PROGRAM GL1_Transfer_Traverse
VAR
	TON_GL1_MTR: TON; // MOTOR FAULT DELAY TIMER
	GL1_MTR: sClearPath;
	GL1_Pulses: INT; // CURRENT PULSE COUNT VALUE
	GL1_Pulse_Counter: CTU; // GL1 MOTOR PULSE COUNTER
	TEST: BOOL;
	GL1_RD: SRoll_Door;
	GL1_PULSE_RESET : BOOL; // RESET THE PULSE COUNTER WHEN COUNTER REACHES PRESET VALUE
	RUN_FWD_TO_GL6_BIT : BOOL; // GL2 OCCUPIED, GL6 REQUESTING PART, RUN TO GL6 POSITION
	RUN_FWD_TO_GL8_BIT : BOOL; // GL2 OCCUPIED, GL8 REQUESTING PART, RUN TO GL8 POSITION
	RUN_REV_TO_GL5B_BIT : BOOL; //GL2 EMPTY, GL2 REQUESTING PART, RUN TO GL5 POSITION
	FAULT_PRESET_TIME: TIME; // FAULT TIMER PRESET TO MOTOR FAULT. DEFAULT IS 1000mS.
	COUNTER_PRESET: WORD; // MAX COUNT VALUE
	TON_GL1_MTR_DONE: BOOL; // TIMER DONE BIT
	KIRK_BIT: BOOL;
	KIRK_BIT2: BOOL;
	KIRK_BIT3: BOOL;
	HI_SPEED: BOOL; // RUN AT HI SPPED TILL FIRST PROX SEEN
	CREEP_SPEED: BOOL; // RUN AT CREEP SPEED TILL SECOND PROX SEEN
	PROX_1_SEEN_AT_GL6: BOOL; // FIRST PROX MADE
	PROX_2_SEEN_AT_GL6: BOOL; // SECOND PROX MADE
	PROX_1_SEEN_AT_GL8: BOOL; // FIRST PROX MADE
	PROX_2_SEEN_AT_GL8: BOOL; // SECOND PROX MADE
	PROX_1_SEEN_AT_GL5B: BOOL; // FIRST PROX MADE
	PROX_2_SEEN_AT_GL5B: BOOL; // SECOND PROX MADE
	TON_CREEP_DELAY: TON; // DELAY CREEP SPEED
	GL6_ENTRY_FTRIG:  F_TRIG;
	GL8_ENTRY_FTRIG:  F_TRIG;
	SwitchFaultTimer: ton;
	SwitchFault: BOOL;
	SwitchTimeElapsed: TIME;
	
END_VAR
VAR // added by the converter: edge detectors and wires of the graphical bodies
    _rt1, _rt2 : R_TRIG;
    _w1, _w2, _w3, _w4, _w5, _w6 : BOOL;
END_VAR

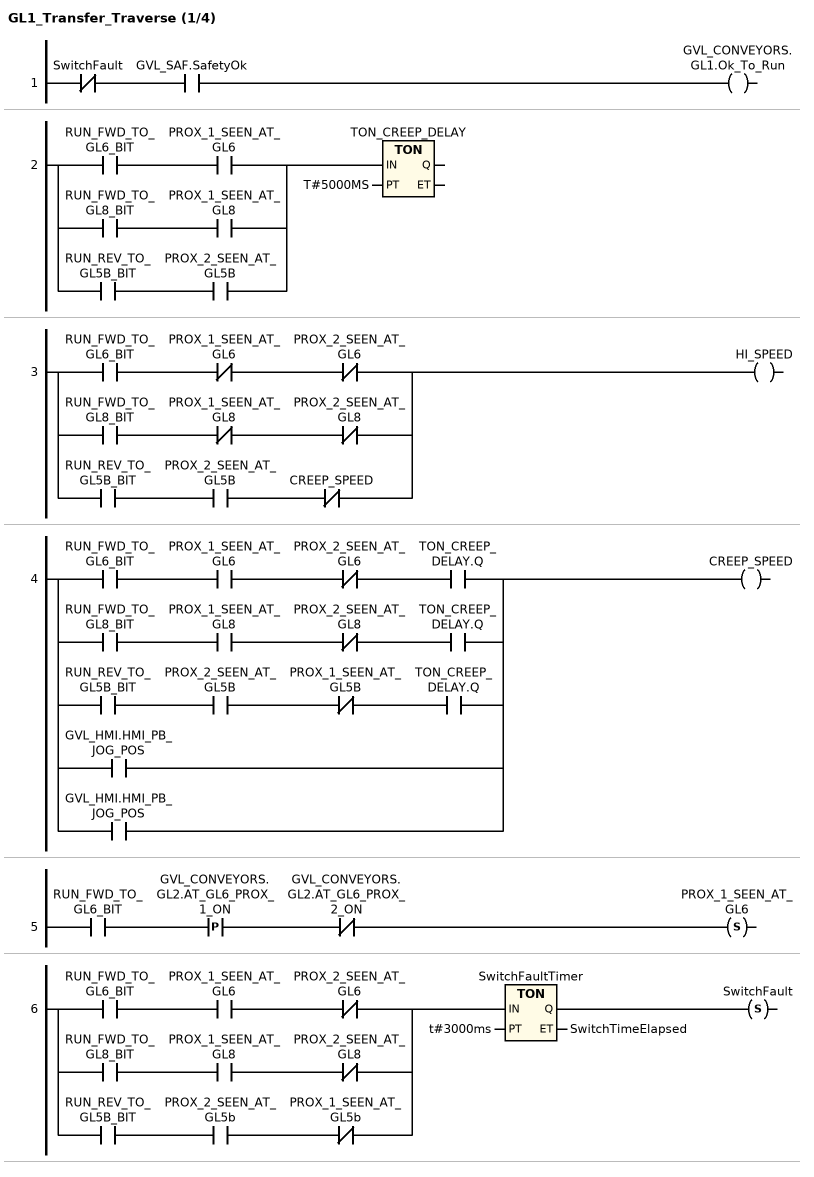
// NETWORK 1
GVL_CONVEYORS.GL1.Ok_To_Run := NOT SwitchFault AND GVL_SAF.SafetyOk;

// NETWORK 2
TON_CREEP_DELAY(IN := RUN_FWD_TO_GL6_BIT AND PROX_1_SEEN_AT_GL6 OR RUN_FWD_TO_GL8_BIT AND PROX_1_SEEN_AT_GL8 OR RUN_REV_TO_GL5B_BIT AND PROX_2_SEEN_AT_GL5B, PT := T#5000MS); // TON

// NETWORK 3
HI_SPEED := RUN_FWD_TO_GL6_BIT AND NOT PROX_1_SEEN_AT_GL6 AND NOT PROX_2_SEEN_AT_GL6 OR RUN_FWD_TO_GL8_BIT AND NOT PROX_1_SEEN_AT_GL8 AND NOT PROX_2_SEEN_AT_GL8 OR RUN_REV_TO_GL5B_BIT AND PROX_2_SEEN_AT_GL5B AND NOT CREEP_SPEED;

// NETWORK 4
CREEP_SPEED := RUN_FWD_TO_GL6_BIT AND PROX_1_SEEN_AT_GL6 AND NOT PROX_2_SEEN_AT_GL6 AND TON_CREEP_DELAY.Q OR RUN_FWD_TO_GL8_BIT AND PROX_1_SEEN_AT_GL8 AND NOT PROX_2_SEEN_AT_GL8 AND TON_CREEP_DELAY.Q OR RUN_REV_TO_GL5B_BIT AND PROX_2_SEEN_AT_GL5B AND NOT PROX_1_SEEN_AT_GL5B AND TON_CREEP_DELAY.Q OR GVL_HMI.HMI_PB_JOG_POS OR GVL_HMI.HMI_PB_JOG_POS;

// NETWORK 5
_rt1(CLK := GVL_CONVEYORS.GL2.AT_GL6_PROX_1_ON);
PROX_1_SEEN_AT_GL6 S= RUN_FWD_TO_GL6_BIT AND _rt1.Q AND NOT GVL_CONVEYORS.GL2.AT_GL6_PROX_2_ON;

// NETWORK 6
SwitchFaultTimer(
    IN := RUN_FWD_TO_GL6_BIT AND PROX_1_SEEN_AT_GL6 AND NOT PROX_2_SEEN_AT_GL6 OR RUN_FWD_TO_GL8_BIT AND PROX_1_SEEN_AT_GL8 AND NOT PROX_2_SEEN_AT_GL8 OR RUN_REV_TO_GL5B_BIT AND PROX_2_SEEN_AT_GL5b AND NOT PROX_1_SEEN_AT_GL5b,
    PT := t#3000ms,
    ET => SwitchTimeElapsed); // TON
SwitchFault S= SwitchFaultTimer.Q;

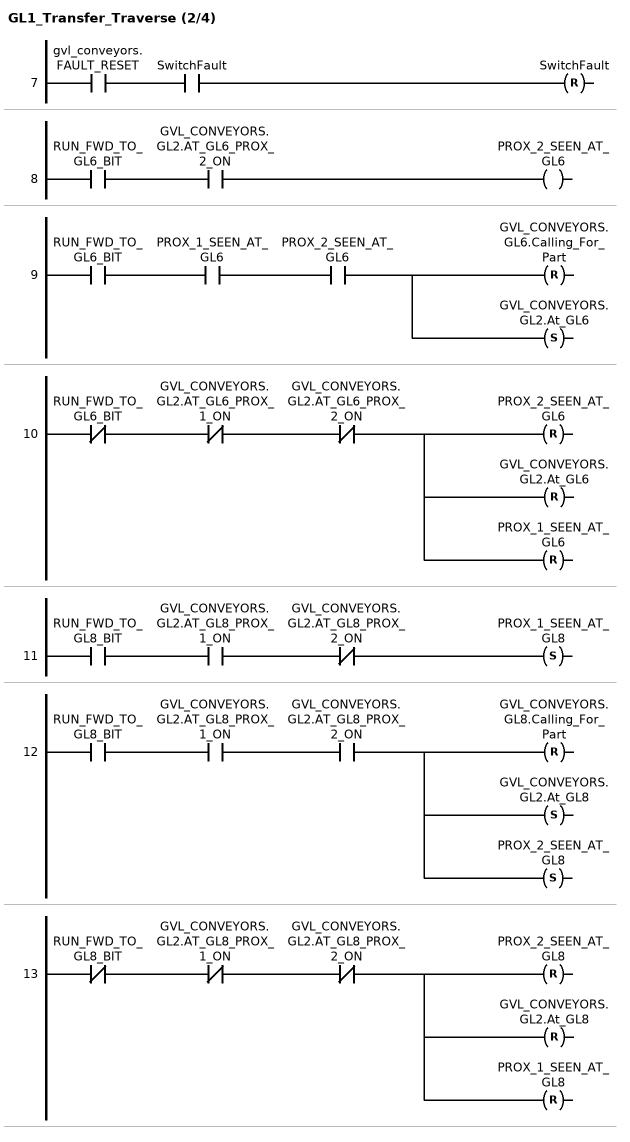
// NETWORK 7
SwitchFault R= gvl_conveyors.FAULT_RESET AND SwitchFault;

// NETWORK 8
PROX_2_SEEN_AT_GL6 := RUN_FWD_TO_GL6_BIT AND GVL_CONVEYORS.GL2.AT_GL6_PROX_2_ON;

// NETWORK 9
_w1 := RUN_FWD_TO_GL6_BIT AND PROX_1_SEEN_AT_GL6 AND PROX_2_SEEN_AT_GL6;
GVL_CONVEYORS.GL6.Calling_For_Part R= _w1;
GVL_CONVEYORS.GL2.At_GL6 S= _w1;

// NETWORK 10
_w2 := NOT RUN_FWD_TO_GL6_BIT AND NOT GVL_CONVEYORS.GL2.AT_GL6_PROX_1_ON AND NOT GVL_CONVEYORS.GL2.AT_GL6_PROX_2_ON;
PROX_2_SEEN_AT_GL6 R= _w2;
GVL_CONVEYORS.GL2.At_GL6 R= _w2;
PROX_1_SEEN_AT_GL6 R= _w2;

// NETWORK 11
PROX_1_SEEN_AT_GL8 S= RUN_FWD_TO_GL8_BIT AND GVL_CONVEYORS.GL2.AT_GL8_PROX_1_ON AND NOT GVL_CONVEYORS.GL2.AT_GL8_PROX_2_ON;

// NETWORK 12
_w3 := RUN_FWD_TO_GL8_BIT AND GVL_CONVEYORS.GL2.AT_GL8_PROX_1_ON AND GVL_CONVEYORS.GL2.AT_GL8_PROX_2_ON;
GVL_CONVEYORS.GL8.Calling_For_Part R= _w3;
GVL_CONVEYORS.GL2.At_GL8 S= _w3;
PROX_2_SEEN_AT_GL8 S= _w3;

// NETWORK 13
_w4 := NOT RUN_FWD_TO_GL8_BIT AND NOT GVL_CONVEYORS.GL2.AT_GL8_PROX_1_ON AND NOT GVL_CONVEYORS.GL2.AT_GL8_PROX_2_ON;
PROX_2_SEEN_AT_GL8 R= _w4;
GVL_CONVEYORS.GL2.At_GL8 R= _w4;
PROX_1_SEEN_AT_GL8 R= _w4;

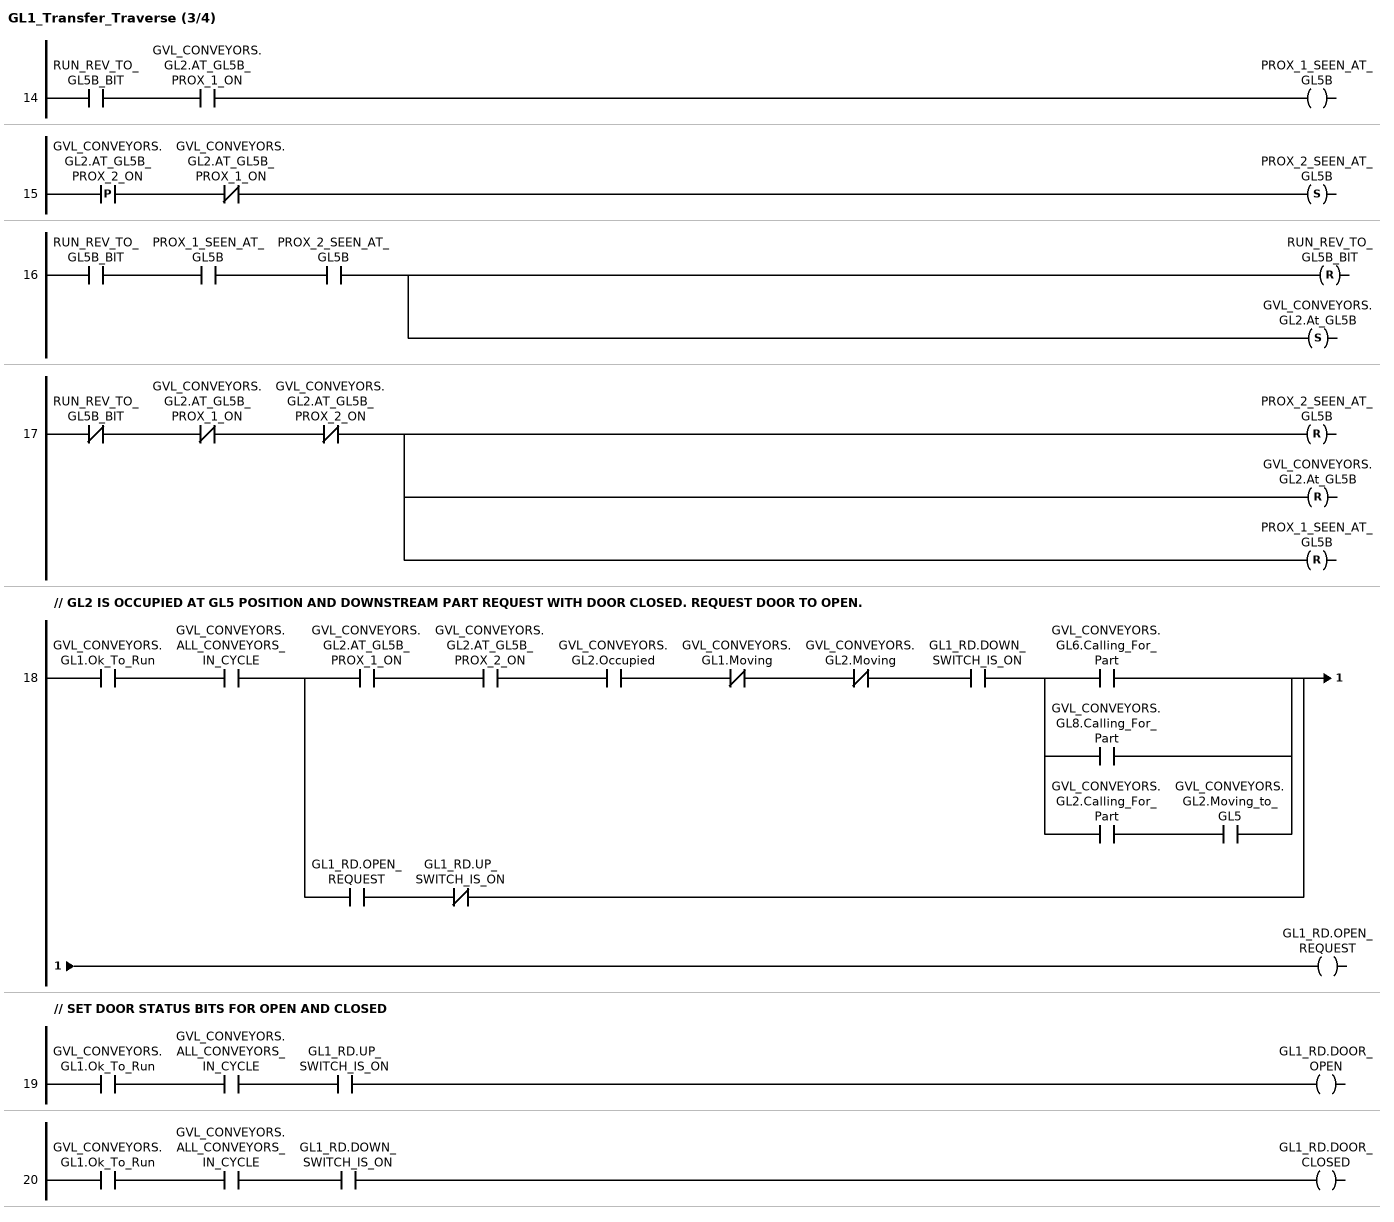
// NETWORK 14
PROX_1_SEEN_AT_GL5B := RUN_REV_TO_GL5B_BIT AND GVL_CONVEYORS.GL2.AT_GL5B_PROX_1_ON;

// NETWORK 15
_rt2(CLK := GVL_CONVEYORS.GL2.AT_GL5B_PROX_2_ON);
PROX_2_SEEN_AT_GL5B S= _rt2.Q AND NOT GVL_CONVEYORS.GL2.AT_GL5B_PROX_1_ON;

// NETWORK 16
_w5 := RUN_REV_TO_GL5B_BIT AND PROX_1_SEEN_AT_GL5B AND PROX_2_SEEN_AT_GL5B;
RUN_REV_TO_GL5B_BIT R= _w5;
GVL_CONVEYORS.GL2.At_GL5B S= _w5;

// NETWORK 17
_w6 := NOT RUN_REV_TO_GL5B_BIT AND NOT GVL_CONVEYORS.GL2.AT_GL5B_PROX_1_ON AND NOT GVL_CONVEYORS.GL2.AT_GL5B_PROX_2_ON;
PROX_2_SEEN_AT_GL5B R= _w6;
GVL_CONVEYORS.GL2.At_GL5B R= _w6;
PROX_1_SEEN_AT_GL5B R= _w6;

// NETWORK 18: // GL2 IS OCCUPIED AT GL5 POSITION AND DOWNSTREAM PART REQUEST WITH DOOR CLOSED. REQUEST DOOR TO OPEN.
GL1_RD.OPEN_REQUEST := GVL_CONVEYORS.GL1.Ok_To_Run AND GVL_CONVEYORS.ALL_CONVEYORS_IN_CYCLE AND (GVL_CONVEYORS.GL2.AT_GL5B_PROX_1_ON AND GVL_CONVEYORS.GL2.AT_GL5B_PROX_2_ON AND GVL_CONVEYORS.GL2.Occupied AND NOT GVL_CONVEYORS.GL1.Moving AND NOT GVL_CONVEYORS.GL2.Moving AND GL1_RD.DOWN_SWITCH_IS_ON AND (GVL_CONVEYORS.GL6.Calling_For_Part OR GVL_CONVEYORS.GL8.Calling_For_Part OR GVL_CONVEYORS.GL2.Calling_For_Part AND GVL_CONVEYORS.GL2.Moving_to_GL5) OR GL1_RD.OPEN_REQUEST AND NOT GL1_RD.UP_SWITCH_IS_ON);

// NETWORK 19: // SET DOOR STATUS BITS FOR OPEN AND CLOSED
GL1_RD.DOOR_OPEN := GVL_CONVEYORS.GL1.Ok_To_Run AND GVL_CONVEYORS.ALL_CONVEYORS_IN_CYCLE AND GL1_RD.UP_SWITCH_IS_ON;

// NETWORK 20
GL1_RD.DOOR_CLOSED := GVL_CONVEYORS.GL1.Ok_To_Run AND GVL_CONVEYORS.ALL_CONVEYORS_IN_CYCLE AND GL1_RD.DOWN_SWITCH_IS_ON;

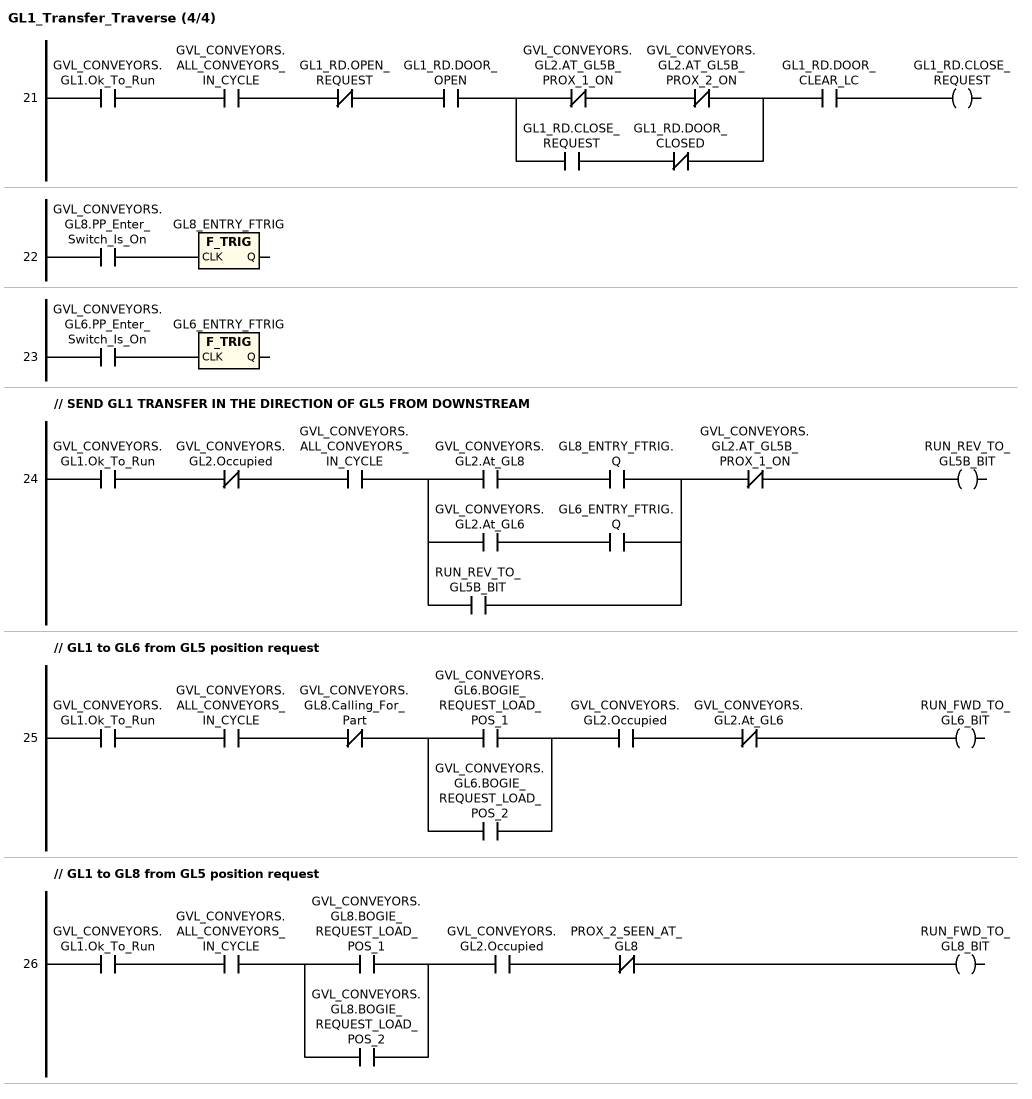
// NETWORK 21
GL1_RD.CLOSE_REQUEST := GVL_CONVEYORS.GL1.Ok_To_Run AND GVL_CONVEYORS.ALL_CONVEYORS_IN_CYCLE AND NOT GL1_RD.OPEN_REQUEST AND GL1_RD.DOOR_OPEN AND (NOT GVL_CONVEYORS.GL2.AT_GL5B_PROX_1_ON AND NOT GVL_CONVEYORS.GL2.AT_GL5B_PROX_2_ON OR GL1_RD.CLOSE_REQUEST AND NOT GL1_RD.DOOR_CLOSED) AND GL1_RD.DOOR_CLEAR_LC;

// NETWORK 22
GL8_ENTRY_FTRIG(CLK := GVL_CONVEYORS.GL8.PP_Enter_Switch_Is_On); // F_TRIG

// NETWORK 23
GL6_ENTRY_FTRIG(CLK := GVL_CONVEYORS.GL6.PP_Enter_Switch_Is_On); // F_TRIG

// NETWORK 24: // SEND GL1 TRANSFER IN THE DIRECTION OF GL5 FROM DOWNSTREAM
RUN_REV_TO_GL5B_BIT := GVL_CONVEYORS.GL1.Ok_To_Run AND NOT GVL_CONVEYORS.GL2.Occupied AND GVL_CONVEYORS.ALL_CONVEYORS_IN_CYCLE AND (GVL_CONVEYORS.GL2.At_GL8 AND GL8_ENTRY_FTRIG.Q OR GVL_CONVEYORS.GL2.At_GL6 AND GL6_ENTRY_FTRIG.Q OR RUN_REV_TO_GL5B_BIT) AND NOT GVL_CONVEYORS.GL2.AT_GL5B_PROX_1_ON;

// NETWORK 25: // GL1 to GL6 from GL5 position request
RUN_FWD_TO_GL6_BIT := GVL_CONVEYORS.GL1.Ok_To_Run AND GVL_CONVEYORS.ALL_CONVEYORS_IN_CYCLE AND NOT GVL_CONVEYORS.GL8.Calling_For_Part AND (GVL_CONVEYORS.GL6.BOGIE_REQUEST_LOAD_POS_1 OR GVL_CONVEYORS.GL6.BOGIE_REQUEST_LOAD_POS_2) AND GVL_CONVEYORS.GL2.Occupied AND NOT GVL_CONVEYORS.GL2.At_GL6;

// NETWORK 26: // GL1 to GL8 from GL5 position request
RUN_FWD_TO_GL8_BIT := GVL_CONVEYORS.GL1.Ok_To_Run AND GVL_CONVEYORS.ALL_CONVEYORS_IN_CYCLE AND (GVL_CONVEYORS.GL8.BOGIE_REQUEST_LOAD_POS_1 OR GVL_CONVEYORS.GL8.BOGIE_REQUEST_LOAD_POS_2) AND GVL_CONVEYORS.GL2.Occupied AND NOT PROX_2_SEEN_AT_GL8;

END_PROGRAM

(* stored: Version 1.1.0.1, ProductVersion 3.1.4024.12
   POU GL1_Transfer_Traverse: Id {009d8071-eb72-437a-a916-da7959eb84a1}, SpecialFunc None *)
